{attribute 'qualified_only'}
VAR_GLOBAL
END_VAR

(* stored: Version 1.1.0.1, ProductVersion 3.1.4024.9
   GVL GVL_RobotArmPickAnadPlaceConstants: Id {5cbc633d-127b-4371-ab70-958a1327469b} *)
